{attribute 'GeneratedUsingTerminal: EL9576-0000-0016'}
{attribute addProperty BoxType "EL9576-0000-0016"}
{attribute addProperty Id "BCT_InputsAT %I*BCT_Inputs_28C1780C15WcStateAT %I*WcState_9091E0EB2InfoDataAT %I*InfoData_32EB74EA10"}
{attribute addProperty CRC "475087744"}
{attribute addProperty Size "27"}
TYPE EL9576_1C514380 EXTENDS EtcSlaveTerminalBase_947E5A46 :
STRUCT
	{attribute addProperty Name "BCT_Inputs"}
	BCT_Inputs : BCT_Inputs_28C1780C;
	{attribute addProperty Name "WcState"}
	WcState : WcState_9091E0EB;
	{attribute addProperty Name "InfoData"}
	InfoData : InfoData_32EB74EA;
END_STRUCT
END_TYPE

(* stored: Version 1.2.0.0, ProductVersion 3.1.4024.9
   DUT EL9576_1C514380: Id {851c1a14-baff-4316-b1f5-8383a2f429c2} *)
